FUNCTION_BLOCK FB_Compressor
VAR_INPUT
END_VAR
VAR_OUTPUT
END_VAR
VAR
END_VAR

END_FUNCTION_BLOCK

(* stored: Version 1.1.0.1, ProductVersion 3.1.4024.10
   POU FB_Compressor: Id {64ad3e54-80e9-4a0f-b456-d3f5d72b18fd}, SpecialFunc None *)
